(* PLC project  *)

FUNCTION ComputeAxis : type
  VAR_INPUT
    speed : REAL;
    mode : INT;
  END_VAR
  VAR_OUTPUT
    errorCode : INT;
  END_VAR

            
// Numeric CASE branches: calls inside branches must become call edges
CASE mode OF
  1:
    ComputeAxis := Scale(speed, 2.0);
  2..5:
    ComputeAxis := Hold(speed);
ELSE
  ComputeAxis := 0.0;
END_CASE;

          
END_FUNCTION

FUNCTION ReadSensor : DINT
  VAR_INPUT
    channel : INT;
  END_VAR
  VAR_IN_OUT
    rawBuffer : TRAFFIC_STATE;
  END_VAR

            
STEP1:
ReadSensor := channel;
ReadSensor := Scale(ReadSensor, rawBuffer);
IF ReadSensor > 100 THEN
  JMP STEP1;
END_IF;

          
END_FUNCTION
